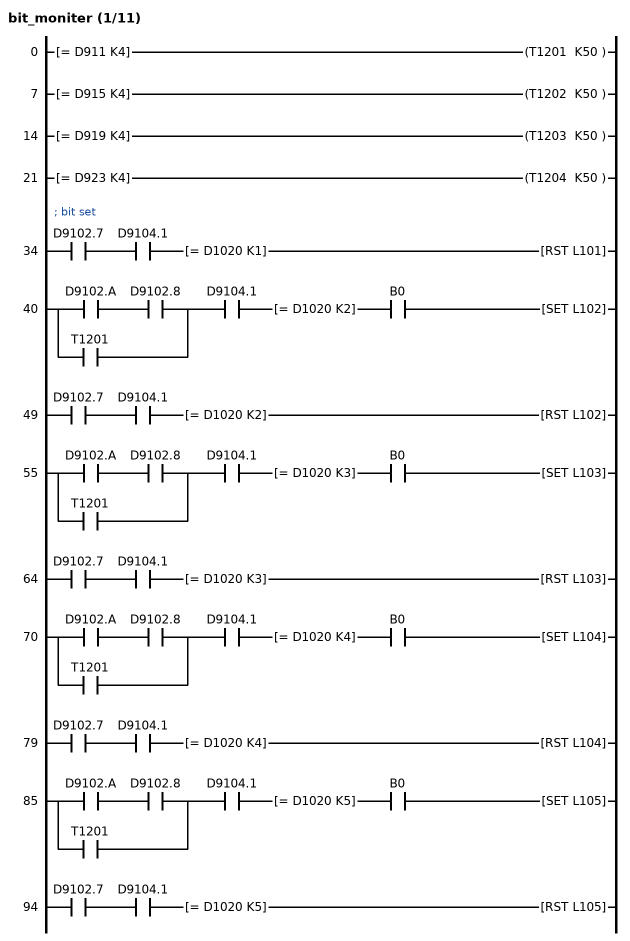
[picture p24: ladder of bit_moniter, rungs at steps 0 to 94]
0     LD=     D911 K4
      OUT     T1201 K50
7     LD=     D915 K4
      OUT     T1202 K50
14    LD=     D919 K4
      OUT     T1203 K50
21    LD=     D923 K4
      OUT     T1204 K50
; bit set
34    LD      D9102.7
      AND     D9104.1
      AND=    D1020 K1
      RST     L101
40    LD      D9102.A
      AND     D9102.8
      OR      T1201
      AND     D9104.1
      AND=    D1020 K2
      AND     B0
      SET     L102
49    LD      D9102.7
      AND     D9104.1
      AND=    D1020 K2
      RST     L102
55    LD      D9102.A
      AND     D9102.8
      OR      T1201
      AND     D9104.1
      AND=    D1020 K3
      AND     B0
      SET     L103
64    LD      D9102.7
      AND     D9104.1
      AND=    D1020 K3
      RST     L103
70    LD      D9102.A
      AND     D9102.8
      OR      T1201
      AND     D9104.1
      AND=    D1020 K4
      AND     B0
      SET     L104
79    LD      D9102.7
      AND     D9104.1
      AND=    D1020 K4
      RST     L104
85    LD      D9102.A
      AND     D9102.8
      OR      T1201
      AND     D9104.1
      AND=    D1020 K5
      AND     B0
      SET     L105
94    LD      D9102.7
      AND     D9104.1
      AND=    D1020 K5
      RST     L105
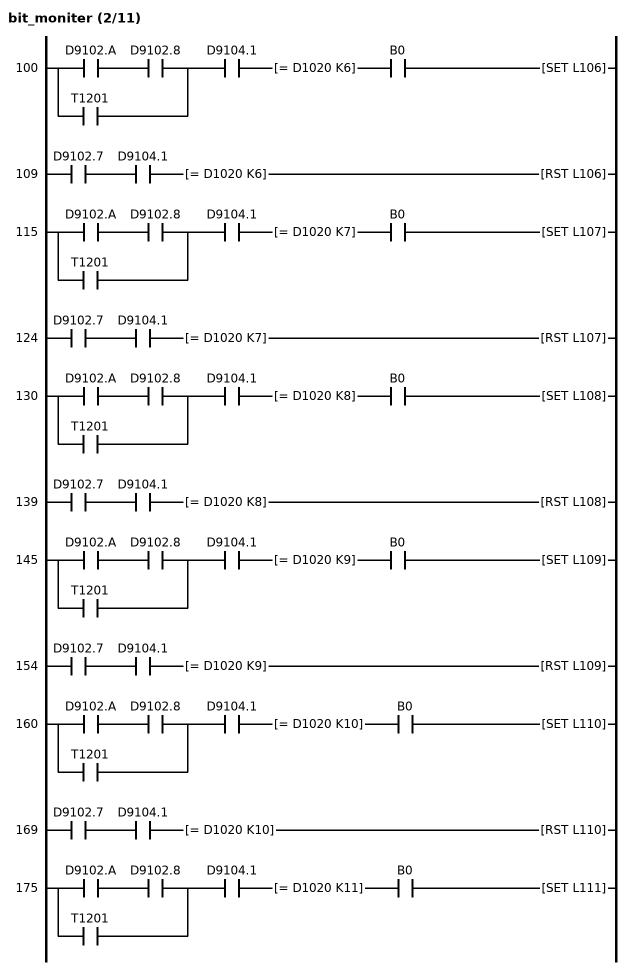
100   LD      D9102.A
      AND     D9102.8
      OR      T1201
      AND     D9104.1
      AND=    D1020 K6
      AND     B0
      SET     L106
109   LD      D9102.7
      AND     D9104.1
      AND=    D1020 K6
      RST     L106
115   LD      D9102.A
      AND     D9102.8
      OR      T1201
      AND     D9104.1
      AND=    D1020 K7
      AND     B0
      SET     L107
124   LD      D9102.7
      AND     D9104.1
      AND=    D1020 K7
      RST     L107
130   LD      D9102.A
      AND     D9102.8
      OR      T1201
      AND     D9104.1
      AND=    D1020 K8
      AND     B0
      SET     L108
139   LD      D9102.7
      AND     D9104.1
      AND=    D1020 K8
      RST     L108
145   LD      D9102.A
      AND     D9102.8
      OR      T1201
      AND     D9104.1
      AND=    D1020 K9
      AND     B0
      SET     L109
154   LD      D9102.7
      AND     D9104.1
      AND=    D1020 K9
      RST     L109
160   LD      D9102.A
      AND     D9102.8
      OR      T1201
      AND     D9104.1
      AND=    D1020 K10
      AND     B0
      SET     L110
169   LD      D9102.7
      AND     D9104.1
      AND=    D1020 K10
      RST     L110
175   LD      D9102.A
      AND     D9102.8
      OR      T1201
      AND     D9104.1
      AND=    D1020 K11
      AND     B0
      SET     L111
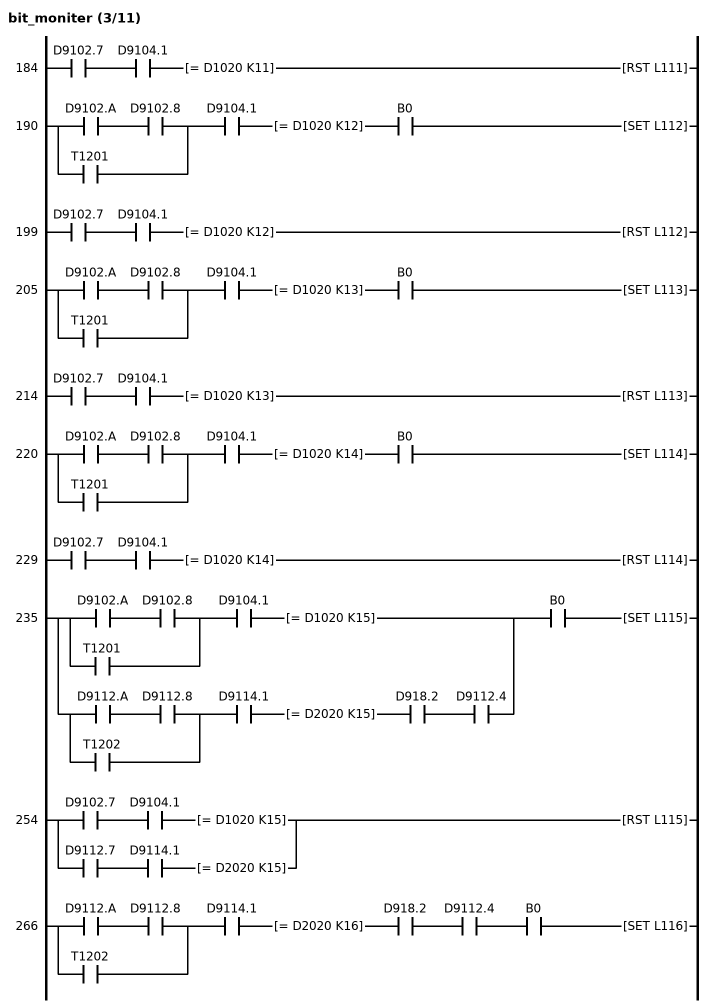
184   LD      D9102.7
      AND     D9104.1
      AND=    D1020 K11
      RST     L111
190   LD      D9102.A
      AND     D9102.8
      OR      T1201
      AND     D9104.1
      AND=    D1020 K12
      AND     B0
      SET     L112
199   LD      D9102.7
      AND     D9104.1
      AND=    D1020 K12
      RST     L112
205   LD      D9102.A
      AND     D9102.8
      OR      T1201
      AND     D9104.1
      AND=    D1020 K13
      AND     B0
      SET     L113
214   LD      D9102.7
      AND     D9104.1
      AND=    D1020 K13
      RST     L113
220   LD      D9102.A
      AND     D9102.8
      OR      T1201
      AND     D9104.1
      AND=    D1020 K14
      AND     B0
      SET     L114
229   LD      D9102.7
      AND     D9104.1
      AND=    D1020 K14
      RST     L114
235   LD      D9102.A
      AND     D9102.8
      OR      T1201
      AND     D9104.1
      AND=    D1020 K15
      LD      D9112.A
      AND     D9112.8
      OR      T1202
      AND     D9114.1
      AND=    D2020 K15
      AND     D918.2
      AND     D9112.4
      ORB
      AND     B0
      SET     L115
254   LD      D9102.7
      AND     D9104.1
      AND=    D1020 K15
      LD      D9112.7
      AND     D9114.1
      AND=    D2020 K15
      ORB
      RST     L115
266   LD      D9112.A
      AND     D9112.8
      OR      T1202
      AND     D9114.1
      AND=    D2020 K16
      AND     D918.2
      AND     D9112.4
      AND     B0
      SET     L116
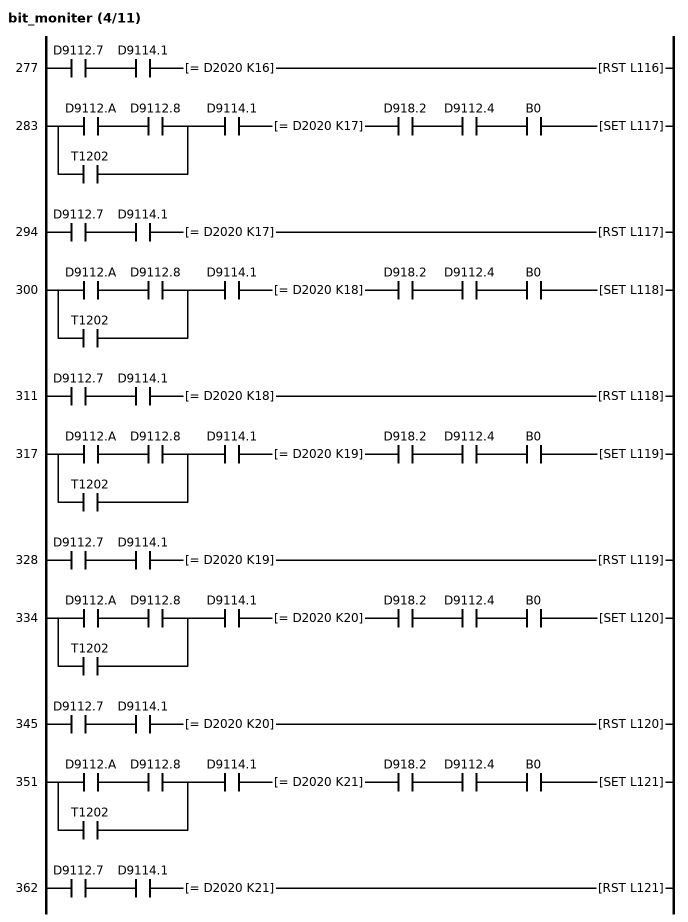
277   LD      D9112.7
      AND     D9114.1
      AND=    D2020 K16
      RST     L116
283   LD      D9112.A
      AND     D9112.8
      OR      T1202
      AND     D9114.1
      AND=    D2020 K17
      AND     D918.2
      AND     D9112.4
      AND     B0
      SET     L117
294   LD      D9112.7
      AND     D9114.1
      AND=    D2020 K17
      RST     L117
300   LD      D9112.A
      AND     D9112.8
      OR      T1202
      AND     D9114.1
      AND=    D2020 K18
      AND     D918.2
      AND     D9112.4
      AND     B0
      SET     L118
311   LD      D9112.7
      AND     D9114.1
      AND=    D2020 K18
      RST     L118
317   LD      D9112.A
      AND     D9112.8
      OR      T1202
      AND     D9114.1
      AND=    D2020 K19
      AND     D918.2
      AND     D9112.4
      AND     B0
      SET     L119
328   LD      D9112.7
      AND     D9114.1
      AND=    D2020 K19
      RST     L119
334   LD      D9112.A
      AND     D9112.8
      OR      T1202
      AND     D9114.1
      AND=    D2020 K20
      AND     D918.2
      AND     D9112.4
      AND     B0
      SET     L120
345   LD      D9112.7
      AND     D9114.1
      AND=    D2020 K20
      RST     L120
351   LD      D9112.A
      AND     D9112.8
      OR      T1202
      AND     D9114.1
      AND=    D2020 K21
      AND     D918.2
      AND     D9112.4
      AND     B0
      SET     L121
362   LD      D9112.7
      AND     D9114.1
      AND=    D2020 K21
      RST     L121
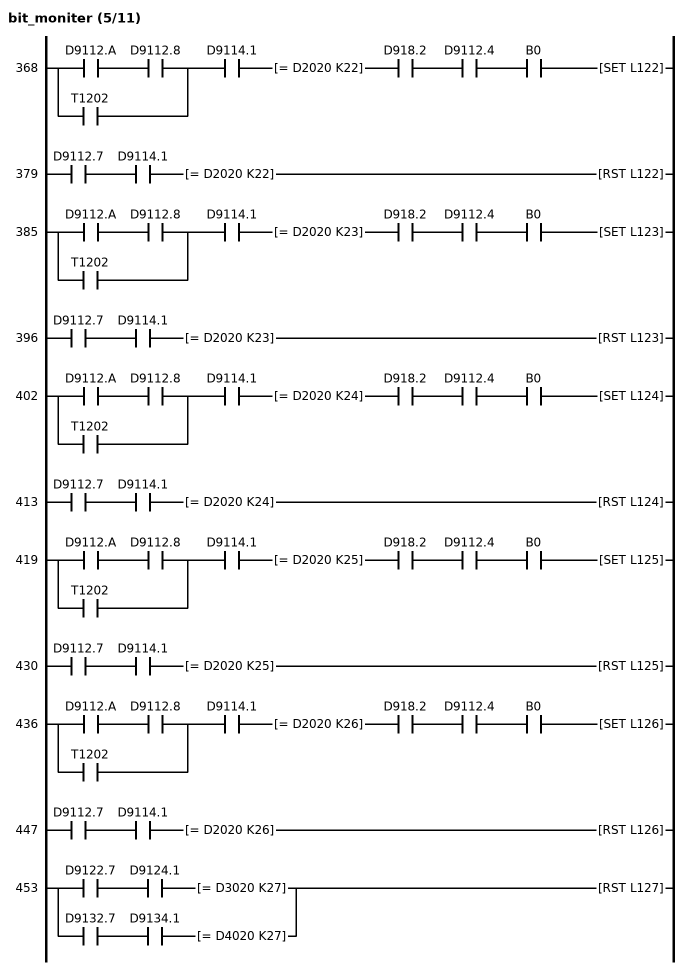
368   LD      D9112.A
      AND     D9112.8
      OR      T1202
      AND     D9114.1
      AND=    D2020 K22
      AND     D918.2
      AND     D9112.4
      AND     B0
      SET     L122
379   LD      D9112.7
      AND     D9114.1
      AND=    D2020 K22
      RST     L122
385   LD      D9112.A
      AND     D9112.8
      OR      T1202
      AND     D9114.1
      AND=    D2020 K23
      AND     D918.2
      AND     D9112.4
      AND     B0
      SET     L123
396   LD      D9112.7
      AND     D9114.1
      AND=    D2020 K23
      RST     L123
402   LD      D9112.A
      AND     D9112.8
      OR      T1202
      AND     D9114.1
      AND=    D2020 K24
      AND     D918.2
      AND     D9112.4
      AND     B0
      SET     L124
413   LD      D9112.7
      AND     D9114.1
      AND=    D2020 K24
      RST     L124
419   LD      D9112.A
      AND     D9112.8
      OR      T1202
      AND     D9114.1
      AND=    D2020 K25
      AND     D918.2
      AND     D9112.4
      AND     B0
      SET     L125
430   LD      D9112.7
      AND     D9114.1
      AND=    D2020 K25
      RST     L125
436   LD      D9112.A
      AND     D9112.8
      OR      T1202
      AND     D9114.1
      AND=    D2020 K26
      AND     D918.2
      AND     D9112.4
      AND     B0
      SET     L126
447   LD      D9112.7
      AND     D9114.1
      AND=    D2020 K26
      RST     L126
453   LD      D9122.7
      AND     D9124.1
      AND=    D3020 K27
      LD      D9132.7
      AND     D9134.1
      AND=    D4020 K27
      ORB
      RST     L127
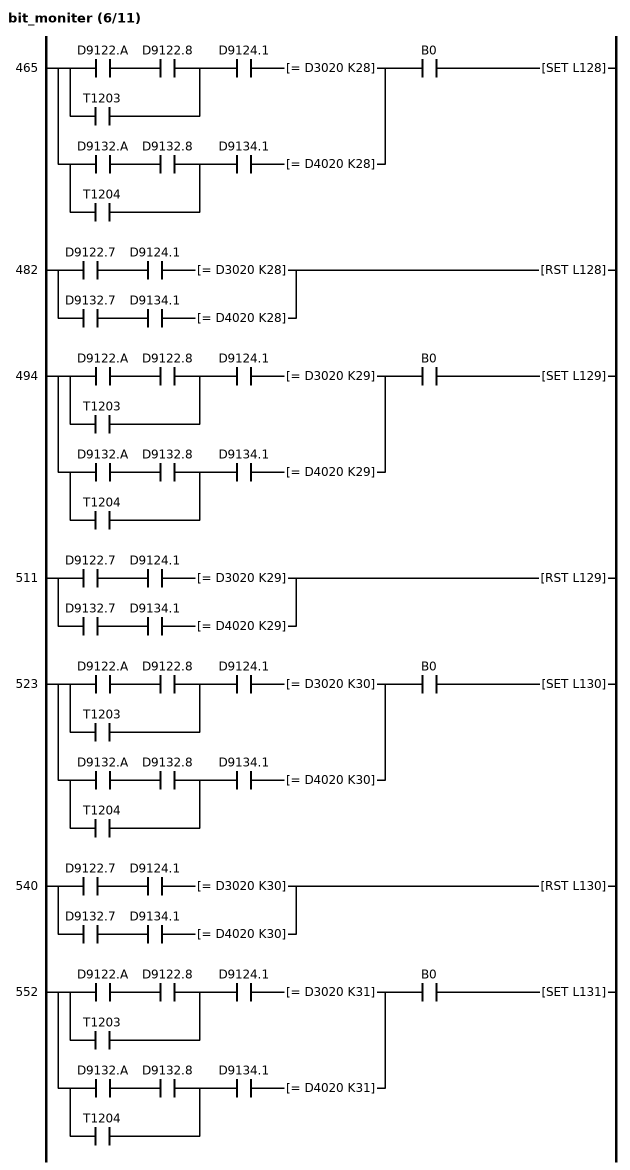
465   LD      D9122.A
      AND     D9122.8
      OR      T1203
      AND     D9124.1
      AND=    D3020 K28
      LD      D9132.A
      AND     D9132.8
      OR      T1204
      AND     D9134.1
      AND=    D4020 K28
      ORB
      AND     B0
      SET     L128
482   LD      D9122.7
      AND     D9124.1
      AND=    D3020 K28
      LD      D9132.7
      AND     D9134.1
      AND=    D4020 K28
      ORB
      RST     L128
494   LD      D9122.A
      AND     D9122.8
      OR      T1203
      AND     D9124.1
      AND=    D3020 K29
      LD      D9132.A
      AND     D9132.8
      OR      T1204
      AND     D9134.1
      AND=    D4020 K29
      ORB
      AND     B0
      SET     L129
511   LD      D9122.7
      AND     D9124.1
      AND=    D3020 K29
      LD      D9132.7
      AND     D9134.1
      AND=    D4020 K29
      ORB
      RST     L129
523   LD      D9122.A
      AND     D9122.8
      OR      T1203
      AND     D9124.1
      AND=    D3020 K30
      LD      D9132.A
      AND     D9132.8
      OR      T1204
      AND     D9134.1
      AND=    D4020 K30
      ORB
      AND     B0
      SET     L130
540   LD      D9122.7
      AND     D9124.1
      AND=    D3020 K30
      LD      D9132.7
      AND     D9134.1
      AND=    D4020 K30
      ORB
      RST     L130
552   LD      D9122.A
      AND     D9122.8
      OR      T1203
      AND     D9124.1
      AND=    D3020 K31
      LD      D9132.A
      AND     D9132.8
      OR      T1204
      AND     D9134.1
      AND=    D4020 K31
      ORB
      AND     B0
      SET     L131
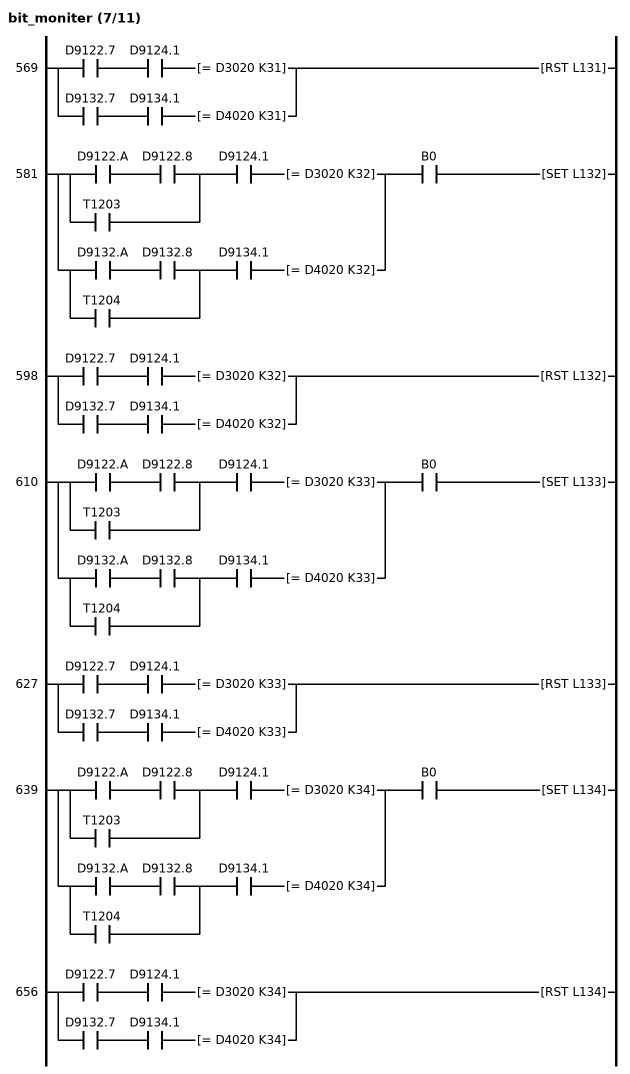
569   LD      D9122.7
      AND     D9124.1
      AND=    D3020 K31
      LD      D9132.7
      AND     D9134.1
      AND=    D4020 K31
      ORB
      RST     L131
581   LD      D9122.A
      AND     D9122.8
      OR      T1203
      AND     D9124.1
      AND=    D3020 K32
      LD      D9132.A
      AND     D9132.8
      OR      T1204
      AND     D9134.1
      AND=    D4020 K32
      ORB
      AND     B0
      SET     L132
598   LD      D9122.7
      AND     D9124.1
      AND=    D3020 K32
      LD      D9132.7
      AND     D9134.1
      AND=    D4020 K32
      ORB
      RST     L132
610   LD      D9122.A
      AND     D9122.8
      OR      T1203
      AND     D9124.1
      AND=    D3020 K33
      LD      D9132.A
      AND     D9132.8
      OR      T1204
      AND     D9134.1
      AND=    D4020 K33
      ORB
      AND     B0
      SET     L133
627   LD      D9122.7
      AND     D9124.1
      AND=    D3020 K33
      LD      D9132.7
      AND     D9134.1
      AND=    D4020 K33
      ORB
      RST     L133
639   LD      D9122.A
      AND     D9122.8
      OR      T1203
      AND     D9124.1
      AND=    D3020 K34
      LD      D9132.A
      AND     D9132.8
      OR      T1204
      AND     D9134.1
      AND=    D4020 K34
      ORB
      AND     B0
      SET     L134
656   LD      D9122.7
      AND     D9124.1
      AND=    D3020 K34
      LD      D9132.7
      AND     D9134.1
      AND=    D4020 K34
      ORB
      RST     L134
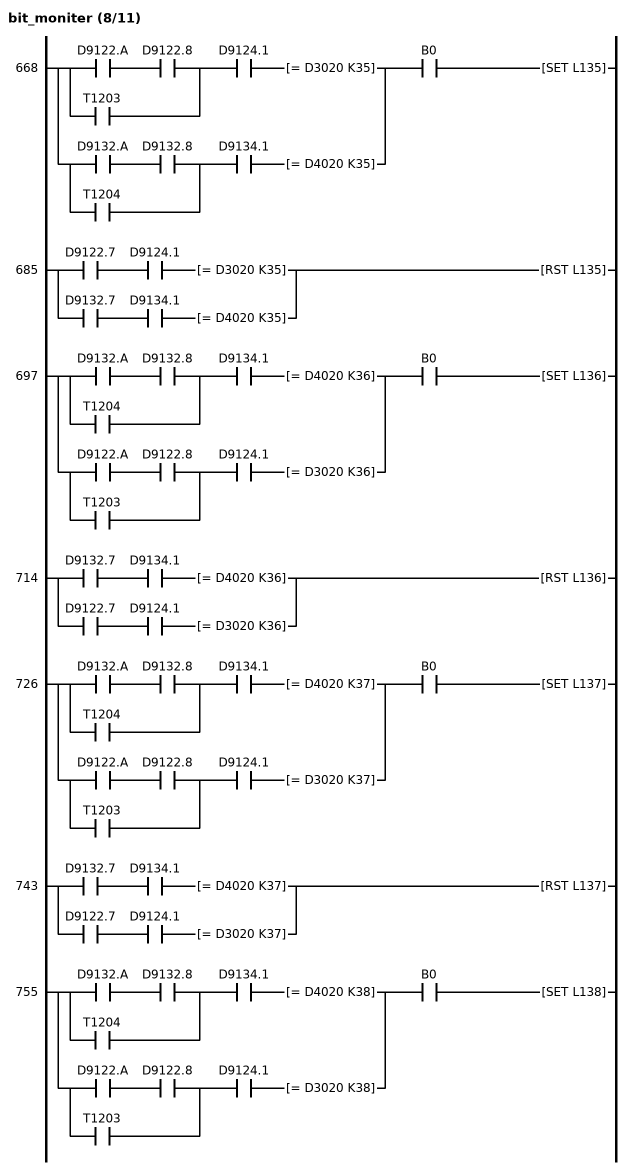
668   LD      D9122.A
      AND     D9122.8
      OR      T1203
      AND     D9124.1
      AND=    D3020 K35
      LD      D9132.A
      AND     D9132.8
      OR      T1204
      AND     D9134.1
      AND=    D4020 K35
      ORB
      AND     B0
      SET     L135
685   LD      D9122.7
      AND     D9124.1
      AND=    D3020 K35
      LD      D9132.7
      AND     D9134.1
      AND=    D4020 K35
      ORB
      RST     L135
697   LD      D9132.A
      AND     D9132.8
      OR      T1204
      AND     D9134.1
      AND=    D4020 K36
      LD      D9122.A
      AND     D9122.8
      OR      T1203
      AND     D9124.1
      AND=    D3020 K36
      ORB
      AND     B0
      SET     L136
714   LD      D9132.7
      AND     D9134.1
      AND=    D4020 K36
      LD      D9122.7
      AND     D9124.1
      AND=    D3020 K36
      ORB
      RST     L136
726   LD      D9132.A
      AND     D9132.8
      OR      T1204
      AND     D9134.1
      AND=    D4020 K37
      LD      D9122.A
      AND     D9122.8
      OR      T1203
      AND     D9124.1
      AND=    D3020 K37
      ORB
      AND     B0
      SET     L137
743   LD      D9132.7
      AND     D9134.1
      AND=    D4020 K37
      LD      D9122.7
      AND     D9124.1
      AND=    D3020 K37
      ORB
      RST     L137
755   LD      D9132.A
      AND     D9132.8
      OR      T1204
      AND     D9134.1
      AND=    D4020 K38
      LD      D9122.A
      AND     D9122.8
      OR      T1203
      AND     D9124.1
      AND=    D3020 K38
      ORB
      AND     B0
      SET     L138
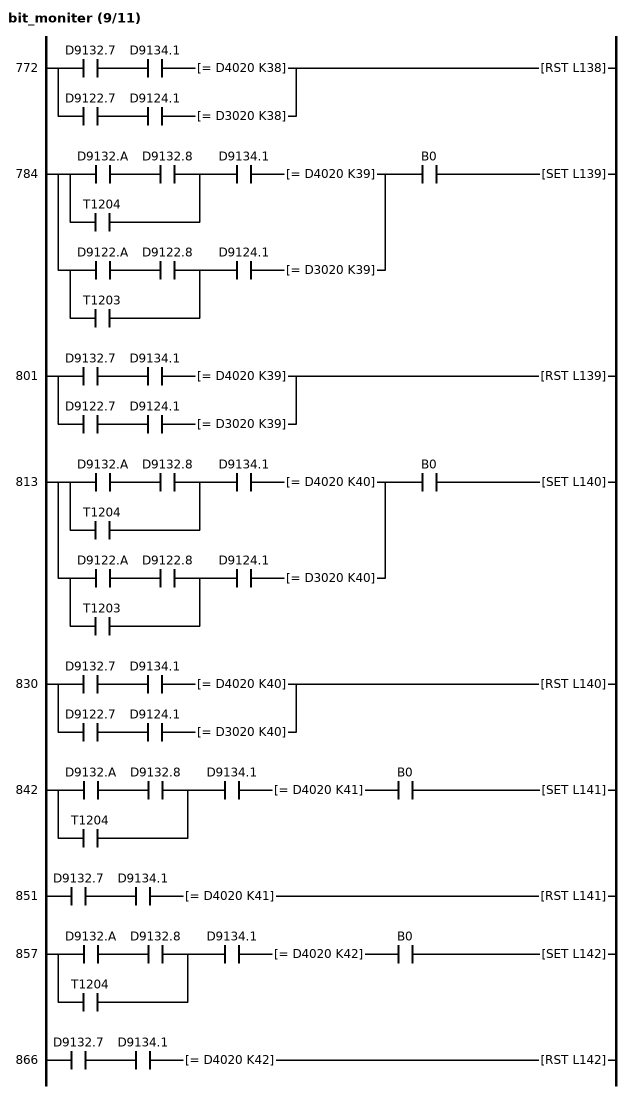
772   LD      D9132.7
      AND     D9134.1
      AND=    D4020 K38
      LD      D9122.7
      AND     D9124.1
      AND=    D3020 K38
      ORB
      RST     L138
784   LD      D9132.A
      AND     D9132.8
      OR      T1204
      AND     D9134.1
      AND=    D4020 K39
      LD      D9122.A
      AND     D9122.8
      OR      T1203
      AND     D9124.1
      AND=    D3020 K39
      ORB
      AND     B0
      SET     L139
801   LD      D9132.7
      AND     D9134.1
      AND=    D4020 K39
      LD      D9122.7
      AND     D9124.1
      AND=    D3020 K39
      ORB
      RST     L139
813   LD      D9132.A
      AND     D9132.8
      OR      T1204
      AND     D9134.1
      AND=    D4020 K40
      LD      D9122.A
      AND     D9122.8
      OR      T1203
      AND     D9124.1
      AND=    D3020 K40
      ORB
      AND     B0
      SET     L140
830   LD      D9132.7
      AND     D9134.1
      AND=    D4020 K40
      LD      D9122.7
      AND     D9124.1
      AND=    D3020 K40
      ORB
      RST     L140
842   LD      D9132.A
      AND     D9132.8
      OR      T1204
      AND     D9134.1
      AND=    D4020 K41
      AND     B0
      SET     L141
851   LD      D9132.7
      AND     D9134.1
      AND=    D4020 K41
      RST     L141
857   LD      D9132.A
      AND     D9132.8
      OR      T1204
      AND     D9134.1
      AND=    D4020 K42
      AND     B0
      SET     L142
866   LD      D9132.7
      AND     D9134.1
      AND=    D4020 K42
      RST     L142
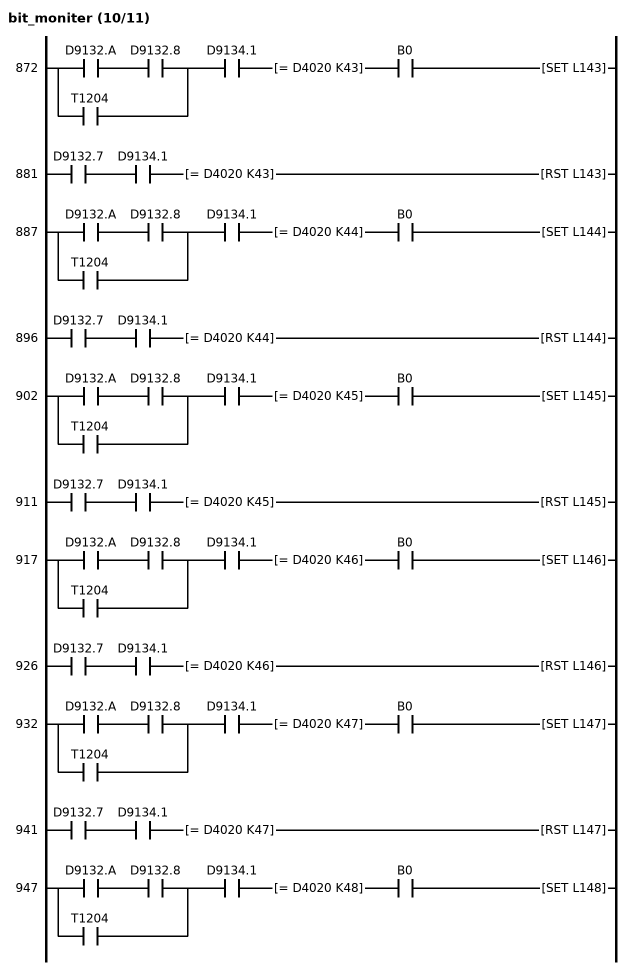
872   LD      D9132.A
      AND     D9132.8
      OR      T1204
      AND     D9134.1
      AND=    D4020 K43
      AND     B0
      SET     L143
881   LD      D9132.7
      AND     D9134.1
      AND=    D4020 K43
      RST     L143
887   LD      D9132.A
      AND     D9132.8
      OR      T1204
      AND     D9134.1
      AND=    D4020 K44
      AND     B0
      SET     L144
896   LD      D9132.7
      AND     D9134.1
      AND=    D4020 K44
      RST     L144
902   LD      D9132.A
      AND     D9132.8
      OR      T1204
      AND     D9134.1
      AND=    D4020 K45
      AND     B0
      SET     L145
911   LD      D9132.7
      AND     D9134.1
      AND=    D4020 K45
      RST     L145
917   LD      D9132.A
      AND     D9132.8
      OR      T1204
      AND     D9134.1
      AND=    D4020 K46
      AND     B0
      SET     L146
926   LD      D9132.7
      AND     D9134.1
      AND=    D4020 K46
      RST     L146
932   LD      D9132.A
      AND     D9132.8
      OR      T1204
      AND     D9134.1
      AND=    D4020 K47
      AND     B0
      SET     L147
941   LD      D9132.7
      AND     D9134.1
      AND=    D4020 K47
      RST     L147
947   LD      D9132.A
      AND     D9132.8
      OR      T1204
      AND     D9134.1
      AND=    D4020 K48
      AND     B0
      SET     L148
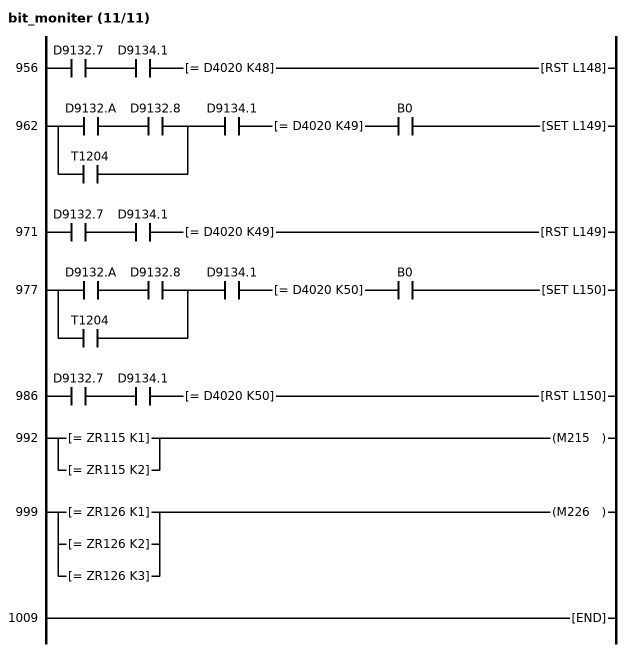
956   LD      D9132.7
      AND     D9134.1
      AND=    D4020 K48
      RST     L148
962   LD      D9132.A
      AND     D9132.8
      OR      T1204
      AND     D9134.1
      AND=    D4020 K49
      AND     B0
      SET     L149
971   LD      D9132.7
      AND     D9134.1
      AND=    D4020 K49
      RST     L149
977   LD      D9132.A
      AND     D9132.8
      OR      T1204
      AND     D9134.1
      AND=    D4020 K50
      AND     B0
      SET     L150
986   LD      D9132.7
      AND     D9134.1
      AND=    D4020 K50
      RST     L150
992   LD=     ZR115 K1
      OR=     ZR115 K2
      OUT     M215
999   LD=     ZR126 K1
      OR=     ZR126 K2
      OR=     ZR126 K3
      OUT     M226
1009  END
END_PROGRAM

FUNCTION_BLOCK c_comm_1
VAR_INPUT
  P1_input : INT;
  P2_input : INT;
  P3_input : INT;
END_VAR
VAR_IN_OUT
  step_on : INT;
END_VAR
VAR_INPUT
  position : INT;
END_VAR
VAR
  p2_buff : INT;
END_VAR
VAR_OUTPUT
  P1_output : INT;
  P2_output : INT;
  P3_output : INT;
END_VAR
VAR_IN_OUT
  end_step_01 : INT;
END_VAR
VAR_OUTPUT
  end_signal : BOOL;
END_VAR
VAR
  mc_1234 : BOOL;
  line1_10_buff : INT;
  line2_10_buff : INT;
END_VAR
VAR_OUTPUT
  next_signal : BOOL;
END_VAR
VAR
  next_signal_01 : BOOL;
  next_signal_03 : BOOL;
  next_signal_04 : BOOL;
  next_signal_05 : BOOL;
  next_signal_06 : BOOL;
  next_signal_07 : BOOL;
  next_signal_08 : BOOL;
  punch1 : BOOL;
  punch3 : BOOL;
  punch4 : BOOL;
  punch5 : BOOL;
  punch6 : BOOL;
  punch7 : BOOL;
END_VAR
VAR_OUTPUT
  punch : BOOL;
END_VAR
VAR
  punch2 : BOOL;
  timee : TIMER;
  tim55 : TIMER;
  timee2 : TIMER;
  timee3 : TIMER;
END_VAR
VAR_INPUT
  d40wait : INT;
END_VAR
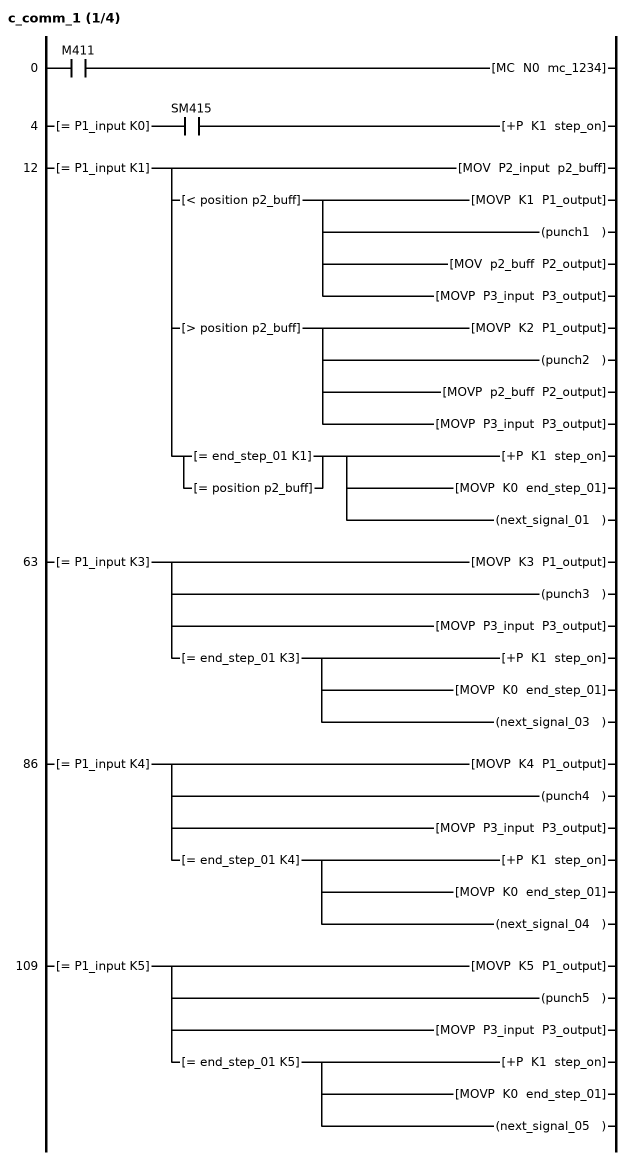
0     LD      M411
      MC      N0 mc_1234
4     LD=     P1_input K0
      AND     SM415
      +P      K1 step_on
12    LD=     P1_input K1
      MOV     P2_input p2_buff
      MPS
      AND<    position p2_buff
      MOVP    K1 P1_output
      OUT     punch1
      MOV     p2_buff P2_output
      MOVP    P3_input P3_output
      MRD
      AND>    position p2_buff
      MOVP    K2 P1_output
      OUT     punch2
      MOVP    p2_buff P2_output
      MOVP    P3_input P3_output
      MPP
      LD=     end_step_01 K1
      OR=     position p2_buff
      ANB
      +P      K1 step_on
      MOVP    K0 end_step_01
      OUT     next_signal_01
63    LD=     P1_input K3
      MOVP    K3 P1_output
      OUT     punch3
      MOVP    P3_input P3_output
      AND=    end_step_01 K3
      +P      K1 step_on
      MOVP    K0 end_step_01
      OUT     next_signal_03
86    LD=     P1_input K4
      MOVP    K4 P1_output
      OUT     punch4
      MOVP    P3_input P3_output
      AND=    end_step_01 K4
      +P      K1 step_on
      MOVP    K0 end_step_01
      OUT     next_signal_04
109   LD=     P1_input K5
      MOVP    K5 P1_output
      OUT     punch5
      MOVP    P3_input P3_output
      AND=    end_step_01 K5
      +P      K1 step_on
      MOVP    K0 end_step_01
      OUT     next_signal_05
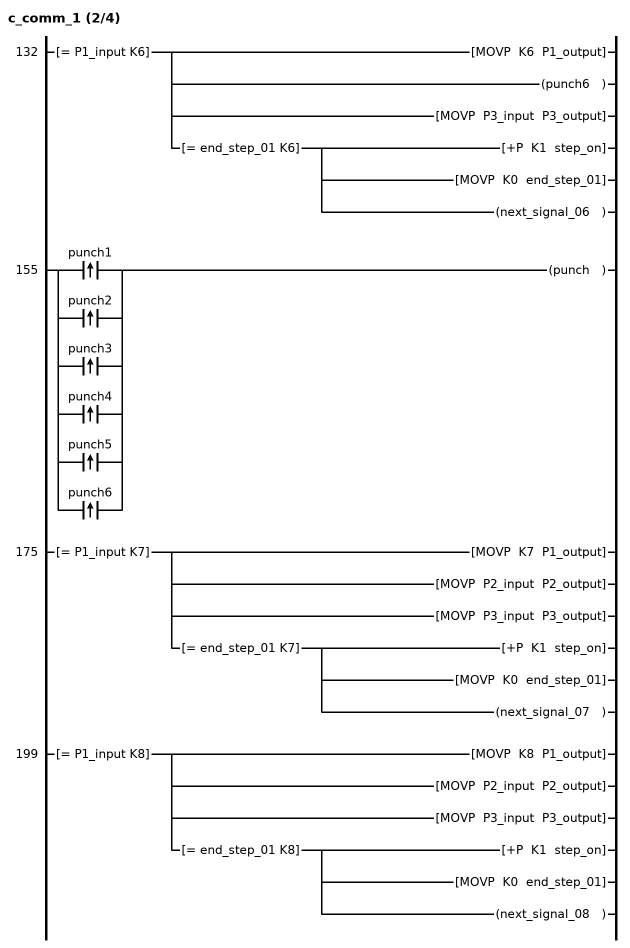
132   LD=     P1_input K6
      MOVP    K6 P1_output
      OUT     punch6
      MOVP    P3_input P3_output
      AND=    end_step_01 K6
      +P      K1 step_on
      MOVP    K0 end_step_01
      OUT     next_signal_06
155   LDP     punch1
      ORP     punch2
      ORP     punch3
      ORP     punch4
      ORP     punch5
      ORP     punch6
      OUT     punch
175   LD=     P1_input K7
      MOVP    K7 P1_output
      MOVP    P2_input P2_output
      MOVP    P3_input P3_output
      AND=    end_step_01 K7
      +P      K1 step_on
      MOVP    K0 end_step_01
      OUT     next_signal_07
199   LD=     P1_input K8
      MOVP    K8 P1_output
      MOVP    P2_input P2_output
      MOVP    P3_input P3_output
      AND=    end_step_01 K8
      +P      K1 step_on
      MOVP    K0 end_step_01
      OUT     next_signal_08
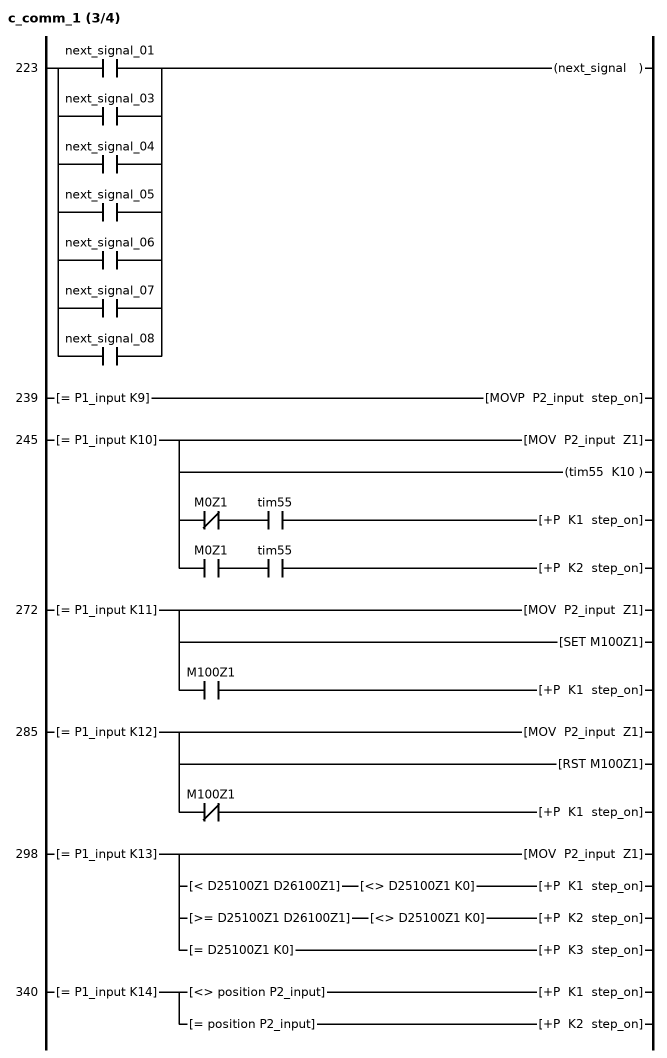
223   LD      next_signal_01
      OR      next_signal_03
      OR      next_signal_04
      OR      next_signal_05
      OR      next_signal_06
      OR      next_signal_07
      OR      next_signal_08
      OUT     next_signal
239   LD=     P1_input K9
      MOVP    P2_input step_on
245   LD=     P1_input K10
      MOV     P2_input Z1
      OUT     tim55 K10
      MPS
      ANI     M0Z1
      AND     tim55
      +P      K1 step_on
      MPP
      AND     M0Z1
      AND     tim55
      +P      K2 step_on
272   LD=     P1_input K11
      MOV     P2_input Z1
      SET     M100Z1
      AND     M100Z1
      +P      K1 step_on
285   LD=     P1_input K12
      MOV     P2_input Z1
      RST     M100Z1
      ANI     M100Z1
      +P      K1 step_on
298   LD=     P1_input K13
      MOV     P2_input Z1
      MPS
      AND<    D25100Z1 D26100Z1
      AND<>   D25100Z1 K0
      +P      K1 step_on
      MRD
      AND>=   D25100Z1 D26100Z1
      AND<>   D25100Z1 K0
      +P      K2 step_on
      MPP
      AND=    D25100Z1 K0
      +P      K3 step_on
340   LD=     P1_input K14
      MPS
      AND<>   position P2_input
      +P      K1 step_on
      MPP
      AND=    position P2_input
      +P      K2 step_on
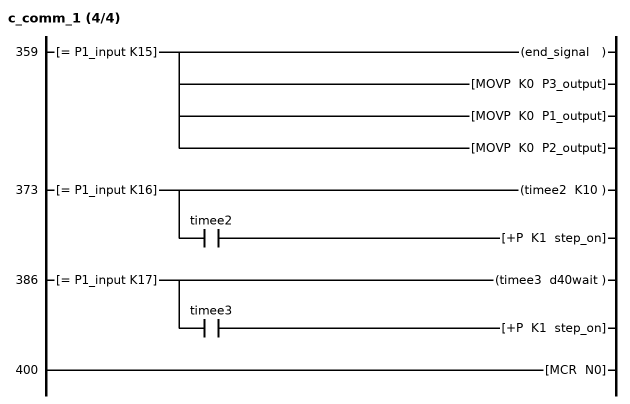
359   LD=     P1_input K15
      OUT     end_signal
      MOVP    K0 P3_output
      MOVP    K0 P1_output
      MOVP    K0 P2_output
373   LD=     P1_input K16
      OUT     timee2 K10
      AND     timee2
      +P      K1 step_on
386   LD=     P1_input K17
      OUT     timee3 d40wait
      AND     timee3
      +P      K1 step_on
400   MCR     N0
END_FUNCTION_BLOCK

FUNCTION_BLOCK c_comm_2
VAR_INPUT
  P1_input : INT;
  P2_input : INT;
  P3_input : INT;
END_VAR
VAR_IN_OUT
  step_on : INT;
END_VAR
VAR_INPUT
  position : INT;
END_VAR
VAR
  p2_buff : INT;
END_VAR
VAR_OUTPUT
  P1_output : INT;
  P2_output : INT;
  P3_output : INT;
END_VAR
VAR_IN_OUT
  end_step_01 : INT;
END_VAR
VAR_OUTPUT
  end_signal : BOOL;
END_VAR
VAR
  mc_1234 : BOOL;
  line1_10_buff : INT;
  line2_10_buff : INT;
END_VAR
VAR_OUTPUT
  next_signal : BOOL;
END_VAR
VAR
  next_signal_01 : BOOL;
  next_signal_03 : BOOL;
  next_signal_04 : BOOL;
  next_signal_05 : BOOL;
  next_signal_06 : BOOL;
  next_signal_07 : BOOL;
  next_signal_08 : BOOL;
  punch1 : BOOL;
  punch3 : BOOL;
  punch4 : BOOL;
  punch5 : BOOL;
  punch6 : BOOL;
  punch7 : BOOL;
END_VAR
VAR_OUTPUT
  punch : BOOL;
END_VAR
VAR
  punch2 : BOOL;
  timee : TIMER;
  tim55 : TIMER;
  timee2 : TIMER;
  timee3 : TIMER;
END_VAR
VAR_INPUT
  d40wait : INT;
END_VAR
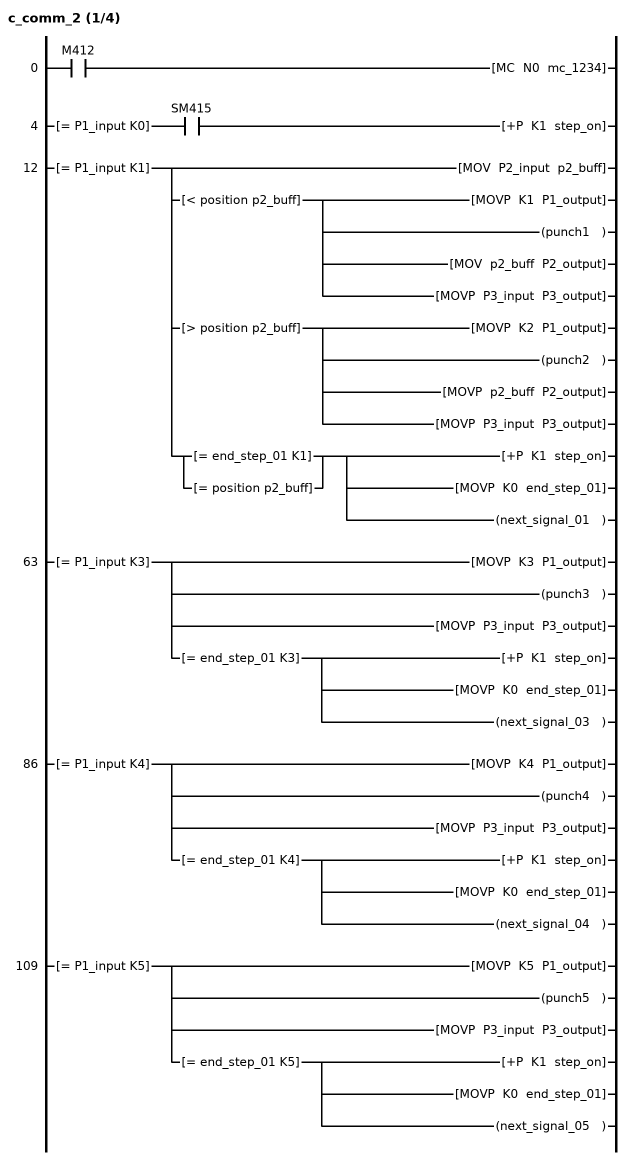
0     LD      M412
      MC      N0 mc_1234
4     LD=     P1_input K0
      AND     SM415
      +P      K1 step_on
12    LD=     P1_input K1
      MOV     P2_input p2_buff
      MPS
      AND<    position p2_buff
      MOVP    K1 P1_output
      OUT     punch1
      MOV     p2_buff P2_output
      MOVP    P3_input P3_output
      MRD
      AND>    position p2_buff
      MOVP    K2 P1_output
      OUT     punch2
      MOVP    p2_buff P2_output
      MOVP    P3_input P3_output
      MPP
      LD=     end_step_01 K1
      OR=     position p2_buff
      ANB
      +P      K1 step_on
      MOVP    K0 end_step_01
      OUT     next_signal_01
63    LD=     P1_input K3
      MOVP    K3 P1_output
      OUT     punch3
      MOVP    P3_input P3_output
      AND=    end_step_01 K3
      +P      K1 step_on
      MOVP    K0 end_step_01
      OUT     next_signal_03
86    LD=     P1_input K4
      MOVP    K4 P1_output
      OUT     punch4
      MOVP    P3_input P3_output
      AND=    end_step_01 K4
      +P      K1 step_on
      MOVP    K0 end_step_01
      OUT     next_signal_04
109   LD=     P1_input K5
      MOVP    K5 P1_output
      OUT     punch5
      MOVP    P3_input P3_output
      AND=    end_step_01 K5
      +P      K1 step_on
      MOVP    K0 end_step_01
      OUT     next_signal_05
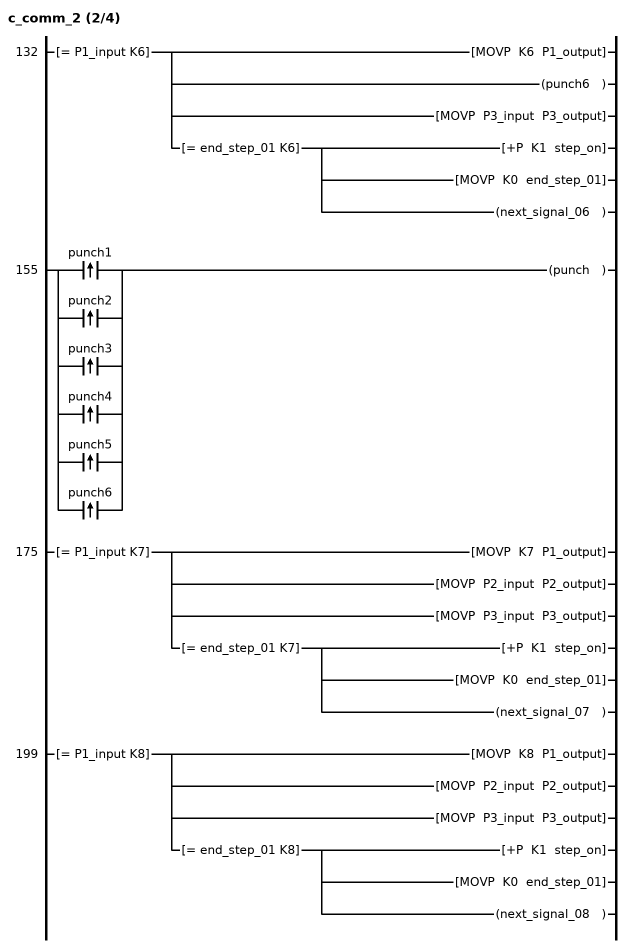
132   LD=     P1_input K6
      MOVP    K6 P1_output
      OUT     punch6
      MOVP    P3_input P3_output
      AND=    end_step_01 K6
      +P      K1 step_on
      MOVP    K0 end_step_01
      OUT     next_signal_06
155   LDP     punch1
      ORP     punch2
      ORP     punch3
      ORP     punch4
      ORP     punch5
      ORP     punch6
      OUT     punch
175   LD=     P1_input K7
      MOVP    K7 P1_output
      MOVP    P2_input P2_output
      MOVP    P3_input P3_output
      AND=    end_step_01 K7
      +P      K1 step_on
      MOVP    K0 end_step_01
      OUT     next_signal_07
199   LD=     P1_input K8
      MOVP    K8 P1_output
      MOVP    P2_input P2_output
      MOVP    P3_input P3_output
      AND=    end_step_01 K8
      +P      K1 step_on
      MOVP    K0 end_step_01
      OUT     next_signal_08
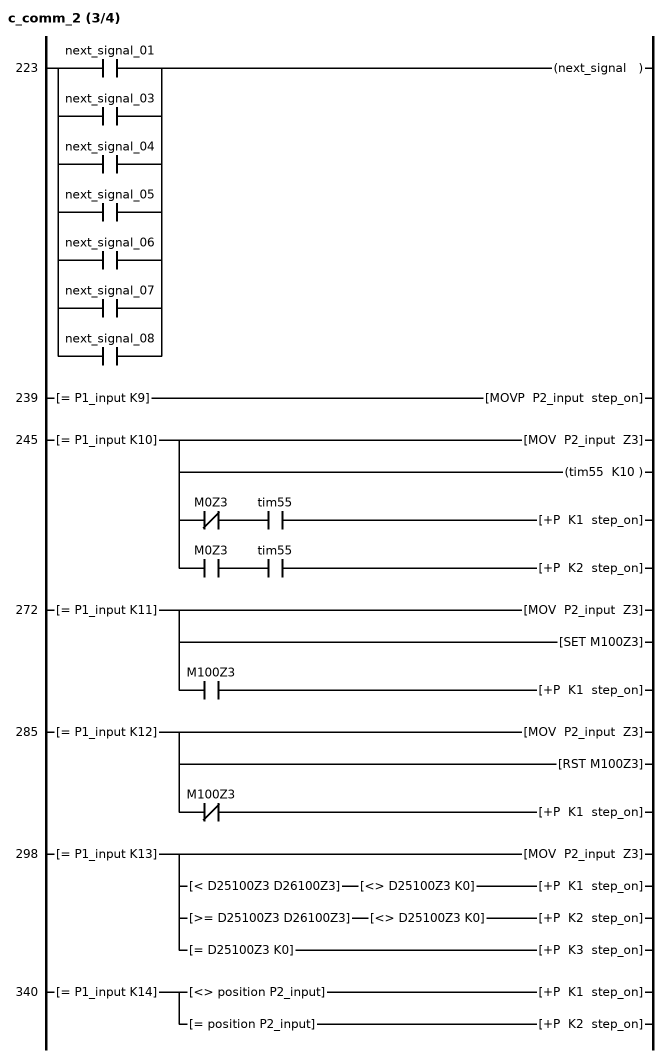
223   LD      next_signal_01
      OR      next_signal_03
      OR      next_signal_04
      OR      next_signal_05
      OR      next_signal_06
      OR      next_signal_07
      OR      next_signal_08
      OUT     next_signal
239   LD=     P1_input K9
      MOVP    P2_input step_on
245   LD=     P1_input K10
      MOV     P2_input Z3
      OUT     tim55 K10
      MPS
      ANI     M0Z3
      AND     tim55
      +P      K1 step_on
      MPP
      AND     M0Z3
      AND     tim55
      +P      K2 step_on
272   LD=     P1_input K11
      MOV     P2_input Z3
      SET     M100Z3
      AND     M100Z3
      +P      K1 step_on
285   LD=     P1_input K12
      MOV     P2_input Z3
      RST     M100Z3
      ANI     M100Z3
      +P      K1 step_on
298   LD=     P1_input K13
      MOV     P2_input Z3
      MPS
      AND<    D25100Z3 D26100Z3
      AND<>   D25100Z3 K0
      +P      K1 step_on
      MRD
      AND>=   D25100Z3 D26100Z3
      AND<>   D25100Z3 K0
      +P      K2 step_on
      MPP
      AND=    D25100Z3 K0
      +P      K3 step_on
340   LD=     P1_input K14
      MPS
      AND<>   position P2_input
      +P      K1 step_on
      MPP
      AND=    position P2_input
      +P      K2 step_on
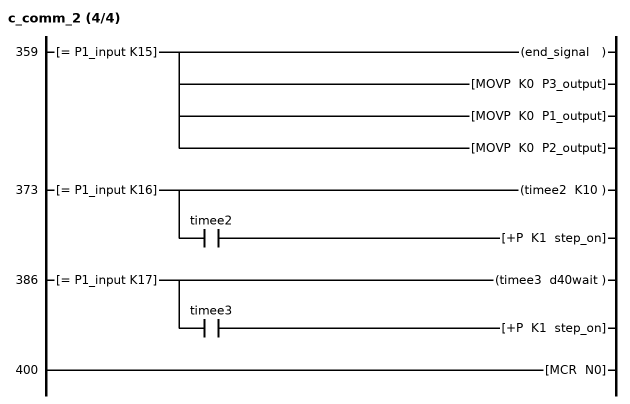
359   LD=     P1_input K15
      OUT     end_signal
      MOVP    K0 P3_output
      MOVP    K0 P1_output
      MOVP    K0 P2_output
373   LD=     P1_input K16
      OUT     timee2 K10
      AND     timee2
      +P      K1 step_on
386   LD=     P1_input K17
      OUT     timee3 d40wait
      AND     timee3
      +P      K1 step_on
400   MCR     N0
END_FUNCTION_BLOCK

FUNCTION_BLOCK c_comm_3
VAR_INPUT
  P1_input : INT;
  P2_input : INT;
  P3_input : INT;
END_VAR
VAR_IN_OUT
  step_on : INT;
END_VAR
VAR_INPUT
  position : INT;
END_VAR
VAR
  p2_buff : INT;
END_VAR
VAR_OUTPUT
  P1_output : INT;
  P2_output : INT;
  P3_output : INT;
END_VAR
VAR_IN_OUT
  end_step_01 : INT;
END_VAR
VAR_OUTPUT
  end_signal : BOOL;
END_VAR
VAR
  mc_1234 : BOOL;
  line1_10_buff : INT;
  line2_10_buff : INT;
END_VAR
VAR_OUTPUT
  next_signal : BOOL;
END_VAR
VAR
  next_signal_01 : BOOL;
  next_signal_03 : BOOL;
  next_signal_04 : BOOL;
  next_signal_05 : BOOL;
  next_signal_06 : BOOL;
  next_signal_07 : BOOL;
  next_signal_08 : BOOL;
  punch1 : BOOL;
  punch3 : BOOL;
  punch4 : BOOL;
  punch5 : BOOL;
  punch6 : BOOL;
  punch7 : BOOL;
END_VAR
VAR_OUTPUT
  punch : BOOL;
END_VAR
VAR
  punch2 : BOOL;
  timee : TIMER;
  tim55 : TIMER;
  timee2 : TIMER;
  timee3 : TIMER;
END_VAR
VAR_INPUT
  d40wait : INT;
END_VAR
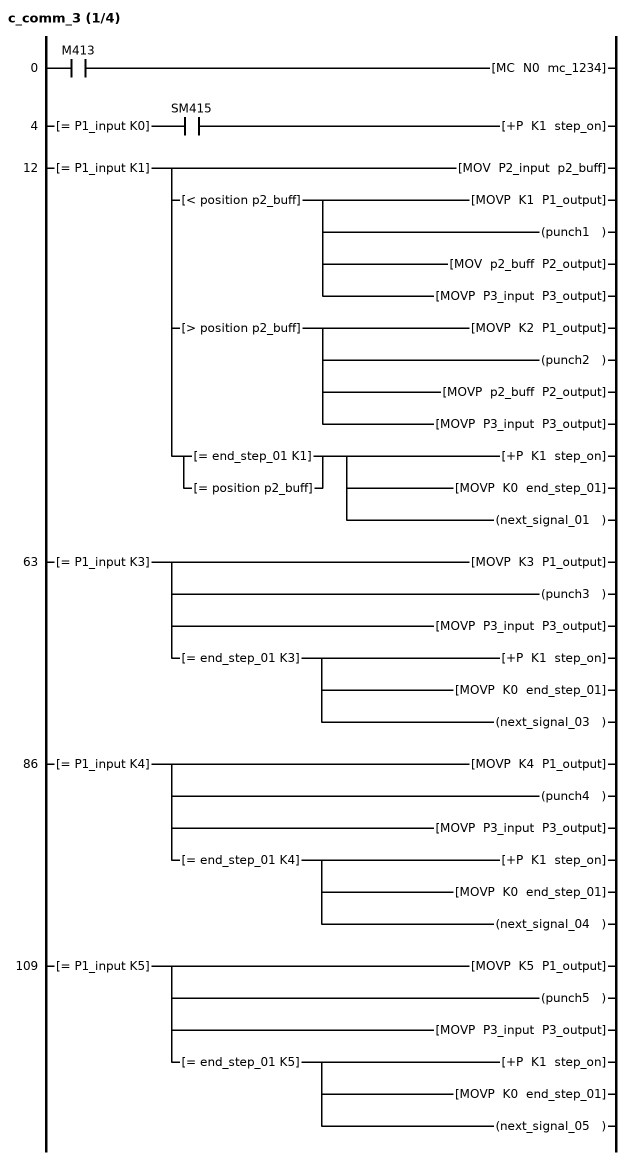
0     LD      M413
      MC      N0 mc_1234
4     LD=     P1_input K0
      AND     SM415
      +P      K1 step_on
12    LD=     P1_input K1
      MOV     P2_input p2_buff
      MPS
      AND<    position p2_buff
      MOVP    K1 P1_output
      OUT     punch1
      MOV     p2_buff P2_output
      MOVP    P3_input P3_output
      MRD
      AND>    position p2_buff
      MOVP    K2 P1_output
      OUT     punch2
      MOVP    p2_buff P2_output
      MOVP    P3_input P3_output
      MPP
      LD=     end_step_01 K1
      OR=     position p2_buff
      ANB
      +P      K1 step_on
      MOVP    K0 end_step_01
      OUT     next_signal_01
63    LD=     P1_input K3
      MOVP    K3 P1_output
      OUT     punch3
      MOVP    P3_input P3_output
      AND=    end_step_01 K3
      +P      K1 step_on
      MOVP    K0 end_step_01
      OUT     next_signal_03
86    LD=     P1_input K4
      MOVP    K4 P1_output
      OUT     punch4
      MOVP    P3_input P3_output
      AND=    end_step_01 K4
      +P      K1 step_on
      MOVP    K0 end_step_01
      OUT     next_signal_04
109   LD=     P1_input K5
      MOVP    K5 P1_output
      OUT     punch5
      MOVP    P3_input P3_output
      AND=    end_step_01 K5
      +P      K1 step_on
      MOVP    K0 end_step_01
      OUT     next_signal_05
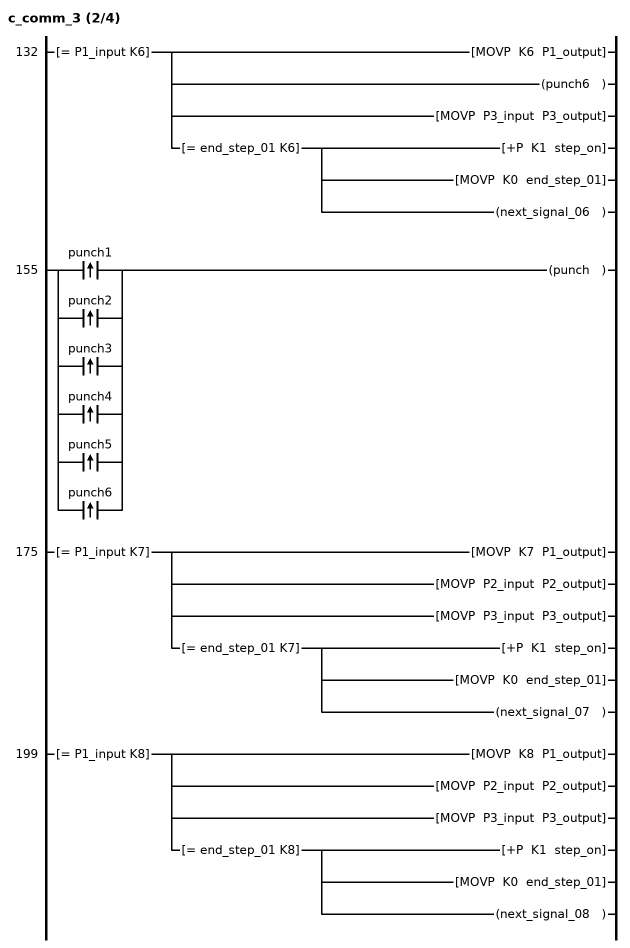
132   LD=     P1_input K6
      MOVP    K6 P1_output
      OUT     punch6
      MOVP    P3_input P3_output
      AND=    end_step_01 K6
      +P      K1 step_on
      MOVP    K0 end_step_01
      OUT     next_signal_06
155   LDP     punch1
      ORP     punch2
      ORP     punch3
      ORP     punch4
      ORP     punch5
      ORP     punch6
      OUT     punch
175   LD=     P1_input K7
      MOVP    K7 P1_output
      MOVP    P2_input P2_output
      MOVP    P3_input P3_output
      AND=    end_step_01 K7
      +P      K1 step_on
      MOVP    K0 end_step_01
      OUT     next_signal_07
199   LD=     P1_input K8
      MOVP    K8 P1_output
      MOVP    P2_input P2_output
      MOVP    P3_input P3_output
      AND=    end_step_01 K8
      +P      K1 step_on
      MOVP    K0 end_step_01
      OUT     next_signal_08
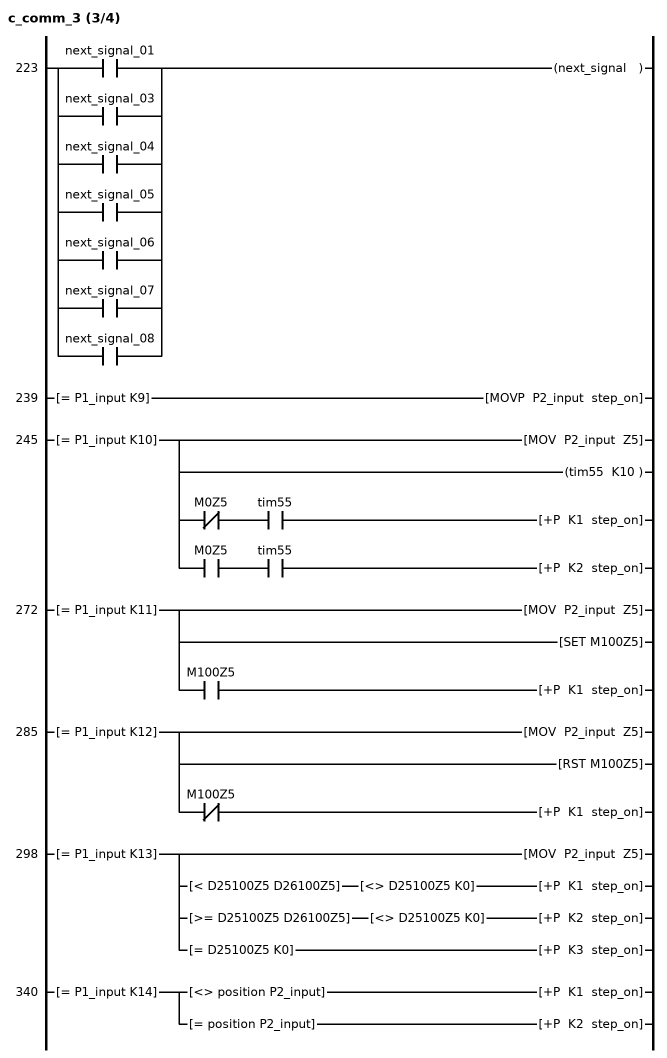
223   LD      next_signal_01
      OR      next_signal_03
      OR      next_signal_04
      OR      next_signal_05
      OR      next_signal_06
      OR      next_signal_07
      OR      next_signal_08
      OUT     next_signal
239   LD=     P1_input K9
      MOVP    P2_input step_on
245   LD=     P1_input K10
      MOV     P2_input Z5
      OUT     tim55 K10
      MPS
      ANI     M0Z5
      AND     tim55
      +P      K1 step_on
      MPP
      AND     M0Z5
      AND     tim55
      +P      K2 step_on
272   LD=     P1_input K11
      MOV     P2_input Z5
      SET     M100Z5
      AND     M100Z5
      +P      K1 step_on
285   LD=     P1_input K12
      MOV     P2_input Z5
      RST     M100Z5
      ANI     M100Z5
      +P      K1 step_on
298   LD=     P1_input K13
      MOV     P2_input Z5
      MPS
      AND<    D25100Z5 D26100Z5
      AND<>   D25100Z5 K0
      +P      K1 step_on
      MRD
      AND>=   D25100Z5 D26100Z5
      AND<>   D25100Z5 K0
      +P      K2 step_on
      MPP
      AND=    D25100Z5 K0
      +P      K3 step_on
340   LD=     P1_input K14
      MPS
      AND<>   position P2_input
      +P      K1 step_on
      MPP
      AND=    position P2_input
      +P      K2 step_on
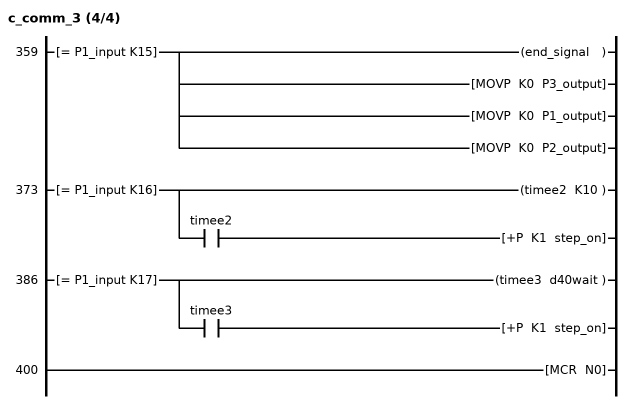
359   LD=     P1_input K15
      OUT     end_signal
      MOVP    K0 P3_output
      MOVP    K0 P1_output
      MOVP    K0 P2_output
373   LD=     P1_input K16
      OUT     timee2 K10
      AND     timee2
      +P      K1 step_on
386   LD=     P1_input K17
      OUT     timee3 d40wait
      AND     timee3
      +P      K1 step_on
400   MCR     N0
END_FUNCTION_BLOCK

FUNCTION_BLOCK c_comm_4
VAR_INPUT
  P1_input : INT;
  P2_input : INT;
  P3_input : INT;
END_VAR
VAR_IN_OUT
  step_on : INT;
END_VAR
VAR_INPUT
  position : INT;
END_VAR
VAR
  p2_buff : INT;
END_VAR
VAR_OUTPUT
  P1_output : INT;
  P2_output : INT;
  P3_output : INT;
END_VAR
VAR_IN_OUT
  end_step_01 : INT;
END_VAR
VAR_OUTPUT
  end_signal : BOOL;
END_VAR
VAR
  mc_1234 : BOOL;
  line1_10_buff : INT;
  line2_10_buff : INT;
END_VAR
VAR_OUTPUT
  next_signal : BOOL;
END_VAR
VAR
  next_signal_01 : BOOL;
  next_signal_03 : BOOL;
  next_signal_04 : BOOL;
  next_signal_05 : BOOL;
  next_signal_06 : BOOL;
  next_signal_07 : BOOL;
  next_signal_08 : BOOL;
  punch1 : BOOL;
  punch3 : BOOL;
  punch4 : BOOL;
  punch5 : BOOL;
  punch6 : BOOL;
  punch7 : BOOL;
END_VAR
VAR_OUTPUT
  punch : BOOL;
END_VAR
VAR
  punch2 : BOOL;
  timee : TIMER;
  tim55 : TIMER;
  timee2 : TIMER;
  timee3 : TIMER;
END_VAR
VAR_INPUT
  d40wait : INT;
END_VAR
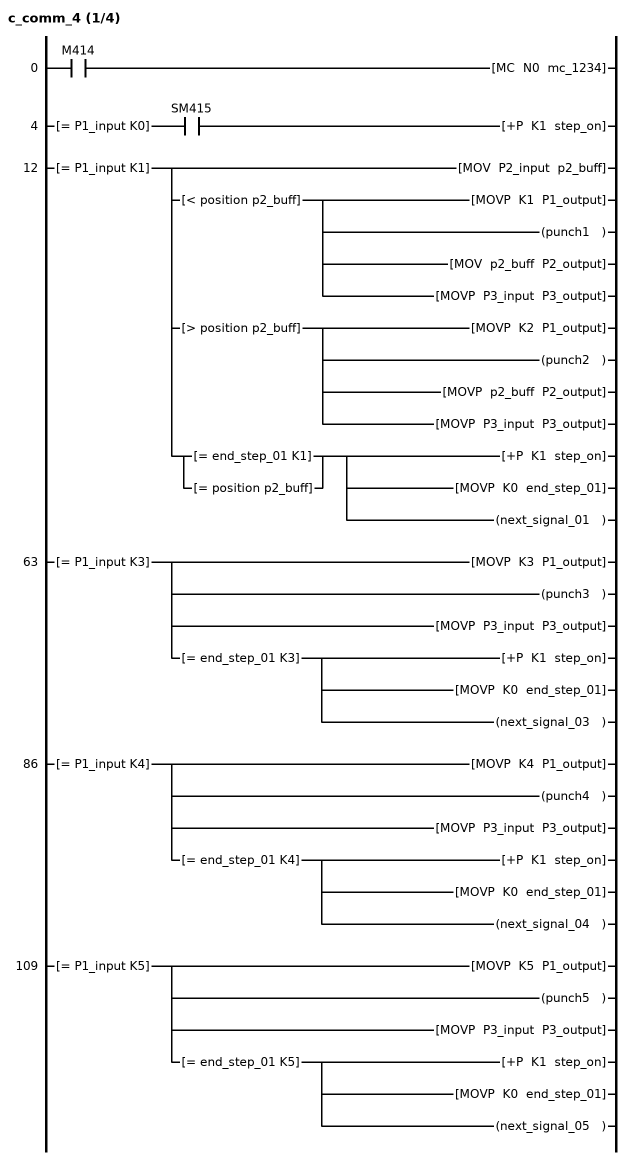
0     LD      M414
      MC      N0 mc_1234
4     LD=     P1_input K0
      AND     SM415
      +P      K1 step_on
12    LD=     P1_input K1
      MOV     P2_input p2_buff
      MPS
      AND<    position p2_buff
      MOVP    K1 P1_output
      OUT     punch1
      MOV     p2_buff P2_output
      MOVP    P3_input P3_output
      MRD
      AND>    position p2_buff
      MOVP    K2 P1_output
      OUT     punch2
      MOVP    p2_buff P2_output
      MOVP    P3_input P3_output
      MPP
      LD=     end_step_01 K1
      OR=     position p2_buff
      ANB
      +P      K1 step_on
      MOVP    K0 end_step_01
      OUT     next_signal_01
63    LD=     P1_input K3
      MOVP    K3 P1_output
      OUT     punch3
      MOVP    P3_input P3_output
      AND=    end_step_01 K3
      +P      K1 step_on
      MOVP    K0 end_step_01
      OUT     next_signal_03
86    LD=     P1_input K4
      MOVP    K4 P1_output
      OUT     punch4
      MOVP    P3_input P3_output
      AND=    end_step_01 K4
      +P      K1 step_on
      MOVP    K0 end_step_01
      OUT     next_signal_04
109   LD=     P1_input K5
      MOVP    K5 P1_output
      OUT     punch5
      MOVP    P3_input P3_output
      AND=    end_step_01 K5
      +P      K1 step_on
      MOVP    K0 end_step_01
      OUT     next_signal_05
